Staubli VAL3: simpleCommTest.dtx

public bool bReceiver
public bool bSender
mdesc mNomSpeed
public num n
public num nB = -1
public num nByteIn[24]
public num nByteOut[24]
public num nTrsfIn[6]
public num nTrsfOut[6]
public sio siTcpReceiver = {link=Socket\Feedback}
public sio siTcpSender = {link=Socket\Motion}
public trsf trShiftIn
public trsf trShiftOut
